TEXTLIST step
  1 = 'Step 1'
  2 = 'Step 2'
  3 = 'Step 3'
  4 = 'Step 4'
  5 = 'Step 5'
  6 = 'Step 6'
  7 = 'Step 7'
  8 = 'Step 8'
  9 = 'Step 9'
  10 = 'Step 10'
  11 = 'Step 11'
  12 = 'Step 12'
  13 = 'Step 13'
  14 = 'Step 14'
  15 = 'Step 15'
  16 = 'Step 16'
  17 = 'Step 17'
  18 = 'Step 18'
  19 = 'Step 19'
  20 = 'Step 20'
  21 = 'Step 21'
  22 = 'Step 22'
  23 = 'Step 23'
  24 = 'Step 24'
  25 = 'Step 25'
  26 = 'Step 26'
  27 = 'Step 27'
  28 = 'Step 28'
  29 = 'Step 29'
  30 = 'Step 30'
   = ''
END_TEXTLIST

(* stored: Version 1.1.0.1, ProductVersion 3.1.4024.11
   TextList step: Id {2ca00dfc-193f-4b94-8840-e7e6c3efff25} *)
